(* CoDeSys 2.3.9.37 project: Cap12_2.pro *)
(* Libraries: Standard.LIB 4.10.05 12:14:46 *)

(* Global variable list: Global_Variables *)
VAR_GLOBAL
  (* Entradas *)
   IW1 : WORD;  (*Variable proveniente del SCADA *)
  (*Salidas*)
   QW1: WORD;  (* Variable a la válvula *)

  (* Otras variables*)
   AperturaValvula: REAL;  (* Valor de ingeniería de apertura de válvula *)
END_VAR

(* POU PLC_PRG, FBD *)
PROGRAM PLC_PRG
VAR
	Escal_Input: Escalado;
	ErrorEscalado: BOOL;
	Escal_Output: Escalado;
END_VAR
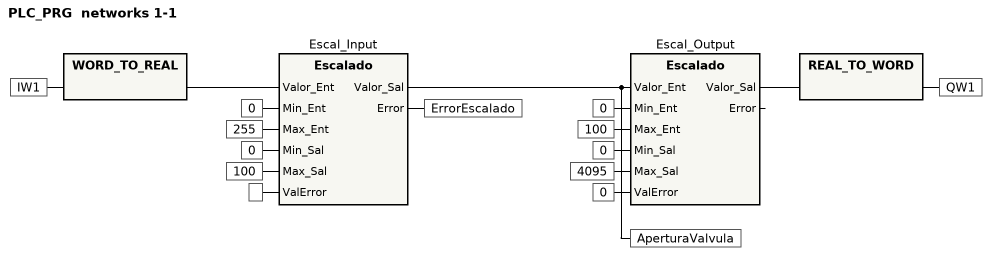
_FBD_ (* Function Block Diagram *)
NETWORK 1
	REAL_TO_WORD(Escal_Output:Escalado(Valor_Ent: <Escal_Input:Escalado(Valor_Ent: WORD_TO_REAL(IW1), Min_Ent: 0, Max_Ent: 255, Min_Sal: 0, Max_Sal: 100, ValError: , Error => ErrorEscalado) => AperturaValvula>, Min_Ent: 0, Max_Ent: 100, Min_Sal: 0, Max_Sal: 4095, ValError: 0)) => QW1
_END_FBD_
END_PROGRAM

(* POU Escalado, ST *)
FUNCTION_BLOCK Escalado
VAR_INPUT
	Valor_Ent : REAL;    (* Valor a convertir *)
	Min_Ent : REAL;      (* Valor mínimo de la entrada *)
	Max_Ent : REAL;	  (* Valor máximo de la entrada *)
	Min_Sal : REAL;      (* Valor mínimo de la salida *)
	Max_Sal : REAL;	   (* . Valor máximo de la salida. *)
       ValError : REAL:=-1;    (*Valor al que poner la salida en caso de error *)
END_VAR
VAR_OUTPUT
	Valor_Sal : REAL;   (*. Valor convertido *)
	Error :  BOOL;         (* Se activa cuando el valor de entrada queda fuera de límites *)
END_VAR
VAR
	pendiente: REAL;
END_VAR
Error:= (Valor_Ent>Max_Ent) OR (Valor_Ent<Min_Ent);

IF NOT Error THEN
   pendiente:=(Max_Sal-Min_Sal)/(Max_Ent-Min_Ent);
   Valor_Sal:=Valor_Ent*pendiente+Min_Sal;
ELSE
   Valor_Sal:=ValError;
END_IF
END_FUNCTION_BLOCK

(* Visualisation Visu
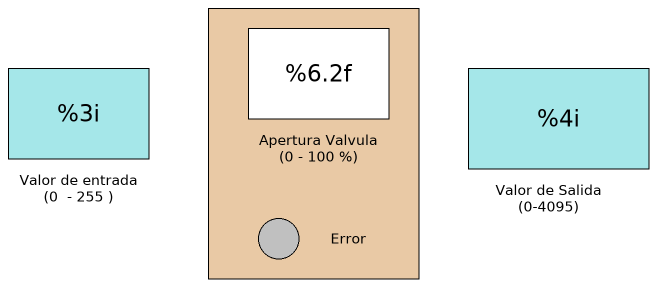
rectangle at (90,100)-(231,191): text "%3i"; shows IW1; editable
rectangle at (50,180)-(271,261): text "Valor de entrada / (0  - 255 )"
rectangle at (330,60)-(471,151): text "%6.2f"; shows AperturaValvula
rectangle at (520,190)-(741,271): text "Valor de Salida / (0-4095)"
ellipse at (340,250)-(381,291): alarm colour if PLC_PRG.ErrorEscalado
rectangle at (370,250)-(491,291): text "Error"
rectangle at (550,100)-(731,201): text "%4i"; shows QW1
rectangle at (290,140)-(511,221): text "Apertura Valvula / (0 - 100 %)"
1 more shapes without text or variables
*)
